KUKA KRL program: chk_w9_grp1_opn.src

&ACCESS RVO4
&COMMENT Axor 903 Z1.1_Z1.2
DEF chk_w9_grp1_opn( )
; Check gripper AXOR 903 OPEN Z1.1/2
;//---- Start User-------

$TIMER[10] = 0
$TIMER_STOP[10] = FALSE

WAIT FOR (NOT $IN[494] AND NOT $IN[496])
WAIT FOR ($IN[493] AND $IN[495])

$TIMER_STOP[10] = TRUE
$TIMER[10] = 0

;//---- End User---------
END
